Fanuc KAREL source: compact_preamble.KL

PROGRAM KB00111
%NOLOCKGROUP
VAR
P1 : FILE
RESULT:INTEGER
BEGIN
RESULT=IO_STATUS(P1)
END KB00111
